# EPICS substitutions: backup/va-x/blvacApp/Db/rga.substitutions
file $(EPICS_BASE)/db/hiden_rga_global.db
{
pattern { Sys		, Dev		, PORT		}
	{ XF:23ID-VA:01	, "{RGA:01}"	, P4	}
}

file $(EPICS_BASE)/db/hiden_rga_bar.db
{
pattern { Sys		, Dev		, PORT		}
 	{ XF:23ID-VA:01	, "{RGA:01}"	, P4	}
}

file $(EPICS_BASE)/db/hiden_rga_prfl.db
{
pattern { Sys		, Dev		, PORT		}
 	{ XF:23ID-VA:01	, "{RGA:01}"	, P4	}
}

file $(EPICS_BASE)/db/hiden_rga_mid.db
{
pattern { Sys		, Dev		, PORT		}
 	{ XF:23ID-VA:01	, "{RGA:01}"	, P4	}
}

file $(EPICS_BASE)/db/hiden_rga_degas.db
{
pattern { Sys		, Dev		, PORT		}
 	{ XF:23ID-VA:01	, "{RGA:01}"	, P4	}
}
